FUNCTION IncNoOverflow : UDINT
VAR_INPUT
	input : UDINT;
END_VAR
VAR
END_VAR

IF input >= 16#FFFFFFFF THEN
	input := 0;
ELSE
	input := input +1;
END_IF

END_FUNCTION

(* stored: Version 1.1.0.1, ProductVersion 3.1.4024.0
   POU IncNoOverflow: Id {d3e498aa-44d1-4c67-8aaa-89b46e344628}, SpecialFunc None *)
